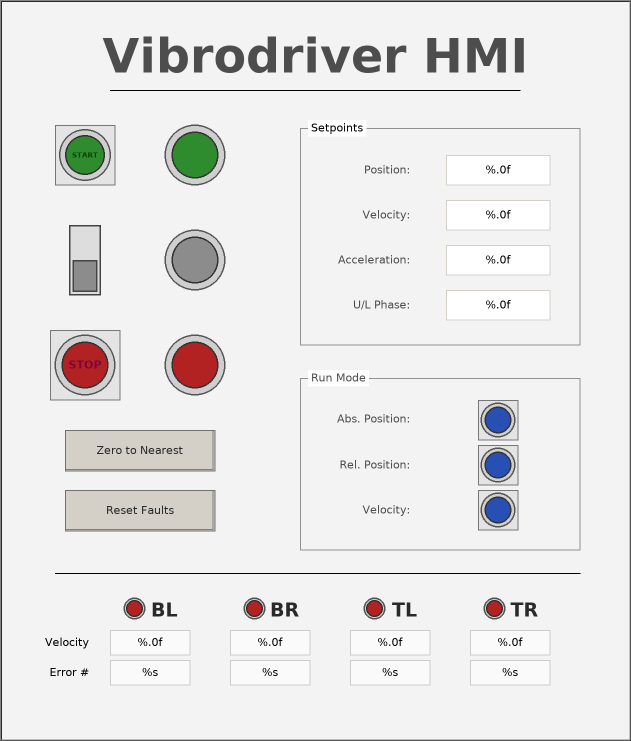
VISUALIZATION hmi  // 631x741
    RoundedRectangle (0,0 631x741)
    PushSwitch (55,125 60x60), tooltip "START", variable: MAIN.bStart, behaviour: TOGGLE, style: Switch-PushSwitch-Green
    Lamp1 (160,120 70x70), variable: MAIN.bStart, style: Lamp-Lamp1-Green
    PushSwitch (50,330 70x70), tooltip "STOP", variable: MAIN.bStop, behaviour: TOGGLE, style: Switch-PushSwitch-Red
    Lamp1 (160,330 70x70), variable: MAIN.bStop, style: Lamp-Lamp1-Red
    GroupBox (300,120 280x225), "Setpoints"
        Label (16,80 97x30), "Velocity:"
        Label (16,125 97x30), "Acceleration:"
        Textfield (146,80 104x30), "%.0f", text variable: MAIN.iVel
            OnMouseClick: write the text variable via InputWithLimits, min -(MAIN.iMaxVel - 200), max MAIN.iMaxVel - 200, format %d
        Textfield (146,35 104x30), "%.0f", text variable: MAIN.iPos
            OnMouseClick: write the text variable via InputWithLimits
        Textfield (146,125 104x30), "%.0f", text variable: MAIN.iAcc
            OnMouseClick: write the text variable via InputWithLimits, min 0, format %d
        Label (16,35 97x30), "Position:"
        Label (16,170 97x30), "U/L Phase:"
        Textfield (146,170 104x30), "%.0f", text variable: MAIN.iPhs
            OnMouseClick: write the text variable via InputWithLimits, min -360, max 360, format %d
    GroupBox (300,370 280x180), "Run Mode"
        Label (16,80 97x30), "Rel. Position:"
        Label (16,125 97x30), "Velocity:"
        Label (16,34 97x30), "Abs. Position:"
        PushSwitch (178,30 40x40), variable: MAIN.bAbsPos, behaviour: TOGGLE, style: Switch-PushSwitch-Blue
        PushSwitch (178,75 40x40), variable: MAIN.bRelPos, behaviour: TOGGLE, style: Switch-PushSwitch-Blue
        PushSwitch (178,120 40x40), variable: MAIN.bVel, behaviour: TOGGLE, style: Switch-PushSwitch-Blue
    DipSwitch (50,225 70x70), tooltip "COUPLE", variable: MAIN.bCouple, behaviour: TOGGLE, style: Switch-DipSwitch-Gray
    Lamp1 (160,225 70x70), variable: MAIN.bCouple, style: Lamp-Lamp1-Gray
    Label (60,350 50x30), "STOP"
    Label (60,140 50x30), "START"
    Button (65,430 150x41), "Zero to Nearest"
        tap MAIN.bZeroNear
    Label (50,20 531x71), "Vibrodriver HMI"
    Line (110,90) (520,90)
    Label (242,590 85x40), "BR"
    Label (362,590 85x40), "TL"
    Label (482,590 85x40), "TR"
    Button (65,490 150x41), "Reset Faults"
        tap MAIN.bResetFaults
    Label (122,590 85x40), "BL"
    Line (55,573) (580,573)
    Lamp1 (122,596 25x25), variable: MAIN.axes[0].Status.Error, style: Lamp-Lamp1-Red
    Lamp1 (242,596 25x25), variable: MAIN.axes[1].Status.Error, style: Lamp-Lamp1-Red
    Lamp1 (482,596 25x25), variable: MAIN.axes[3].Status.Error, style: Lamp-Lamp1-Red
    Lamp1 (362,596 25x25), variable: MAIN.axes[2].Status.Error, style: Lamp-Lamp1-Red
    Textfield (110,630 80x25), "%.0f", text variable: MAIN.axes[0].NcToPlc.ActVelo
    Textfield (230,630 80x25), "%.0f", text variable: MAIN.axes[1].NcToPlc.ActVelo
    Textfield (350,630 80x25), "%.0f", text variable: MAIN.axes[2].NcToPlc.ActVelo
    Textfield (470,630 80x25), "%.0f", text variable: MAIN.axes[3].NcToPlc.ActVelo
    Textfield (110,660 80x25), "%s", text variable: MAIN.arrHexErrors[0]
    Textfield (230,660 80x25), "%s", text variable: MAIN.arrHexErrors[1]
    Textfield (350,660 80x25), "%s", text variable: MAIN.arrHexErrors[2]
    Textfield (470,660 80x25), "%s", text variable: MAIN.arrHexErrors[3]
    Label (40,660 52x25), "Error #"
    Label (40,630 52x25), "Velocity"
END_VISUALIZATION

(* stored: Version 1.1.0.1, ProductVersion 3.1.4024.13
   Visu hmi: Id {871559c6-b0ee-4414-8ee3-84a32fbb96ef} *)
